TYPE SCompensation :
STRUCT
	IsActive: BOOL;	

	(* ID of the Control Primitive that cannot operate anymore. *)
	SickPrimitiveId: UINT;
	
	(* Specifies whether the sick primitive is replaced by another primitive or a sequence. *)
	NewType: EBehaviorType;
	
	(* If NewType is primitive or user-sequence: ID of the sick primitive's replacement. *)
	NewId: UINT;
	
	(* If needed, parameters that are set (or overwritten) before executing the replacement.
	   For replacement types primtive or user-generated sequence, only the first element is used. *)
	ParameterSets: ARRAY [ResiConst.ARR_MIN..ResiConst.MODULE_SEQ_ARR_MAX] OF ParameterSet;
	
	(* If NewType is generated sequence: The (linear) sequence of copmensation primitives. *)
	PrimitiveIds: ARRAY [ResiConst.ARR_MIN..ResiConst.MODULE_SEQ_ARR_MAX] OF UINT;
END_STRUCT
END_TYPE

(* stored: Version 1.1.0.1, ProductVersion 3.1.4024.9
   DUT SCompensation: Id {eaf8ba8f-16d5-45a4-bd8b-bcdad385d8dc} *)
